# EPICS substitutions: wtrvac/Db/vac.substitutions
file "TP_AI.template" { pattern
{P,  		    SIG,	OFFS, TYP,    PREC,   EGU,   LOPR,  HOPR, H,	MAXVAL, PB_ADDR}
{CstatH-Vac:TP001,   MotV,	248,  BYTE,   0,      "V",   0,	100,	100,	100,	5}
{CstatH-Vac:TP001,   BearingT,	249,  BYTE,   0,      "°C",  0,	100,	100,	100,	5}
{CstatH-Vac:TP001,   PSupplyT,	250,  BYTE,   0,      "°C",  0,	100,	100,	100,	5}
{CstatH-Vac:TP001,   CPU_T,	251,  BYTE,   0,      "°C",  0,	100,	100,	100,	5}
{CstatH-Vac:TP001,   MotI,	256,  UINT16, 3,      "A",   0,	10,	10000,	10,	5}
{CstatH-Vac:TP001,   MotP,	258,  UINT16, 0,      "W",   0,	200,	200,	200,	5}
{CstatH-Vac:TP001,   MotPLimit,	260,  UINT16, 0,      "W",   0,	200,	200,	200,	5}
{CstatH-Vac:TP001,   Freq,	262,  UINT16, 0,      "Hz",  0,	1500,	1500,	1500,	5}
{CstatH-Vac:TP001,   FreqSP,	264,  UINT16, 0,      "Hz",  0,	1500,	1500,	1500,	5}
{CstatH-Vac:TP001,   NoOfStarts,266,  UINT16, 0,      "",    0,	65535,	65535,	65535,	5}
{CstatH-Vac:TP001,   LastOnTime,268,  UINT16, 0,      "min.",0,	65535,	65535,	65535,	5}
{CstatH-Vac:TP001,   OpTime,	270,  UINT16, 0,      "h",   0,	65535,	65535,	65535,	5}
}

file "TP_TD20.template" { pattern
{P,  			OFFS,	PB_ADDR}
{CstatH-Vac:TP002,   	278,  	6}
{CstatV-Vac:TP050,   	742,  	8}
{CstatV-Vac:TP060,   	906,  	9}
}

file "CtrlBitwRdBack.template" { pattern

{P,                   SIG,	S_OFFS, S_BIT, S_ZNAM, S_ONAM, C_OFFS, C_BIT, C_ZNAM,   C_ONAM,	INIT_EVNT}
{CstatH-Vac:TP002,    Remote,	276,	 7     Local,  Remote, 46,	  2,	 Local, Remote,	7}
{CstatV-Vac:TP050,    Remote,	740,	 7     Local,  Remote, 144,	  2,	 Local, Remote,	7}
{CstatV-Vac:TP060,    Remote,	904,	 7     Local,  Remote, 194,	  2,	 Local, Remote,	7}
#{CstatH-Vac:TP002,    On,	276,	 2     OFF,    ON,     47,	  0,	 Stop,  Start,	7}
}

file "ArcDet.template" { pattern
{SYS,	SUBS,	DEV,	  SIG,	    OFFS,	BIT,	ZNAM,	ONAM, DESC}
{HPRF,	Distr,	ArcDet01, cmdReset, 98,	0,	Idle,	Reset,	 "Reset Command"}
{HPRF,	Distr,	ArcDet01, cmdTest,  98,	1,	Idle,	Test, 	 "Test Command"}
{HPRF,	Distr,	ArcDet02, cmdReset, 98,	2,	Idle,	Reset,	 "Reset Command"}
{HPRF,	Distr,	ArcDet02, cmdTest,  98,	3,	Idle,	Test, 	 "Test Command"}
{HPRF,	Distr,	ArcDet03, cmdReset, 98,	4,	Idle,	Reset,	 "Reset Command"}
{HPRF,	Distr,	ArcDet03, cmdTest,  98,	5,	Idle,	Test, 	 "Test Command"}
{HPRF,	Distr,	ArcDet04, cmdReset, 98,	6,	Idle,	Reset,	 "Reset Command"}
{HPRF,	Distr,	ArcDet04, cmdTest,  98,	7,	Idle,	Test, 	 "Test Command"}
{HPRF,	Distr,	ArcDet05, cmdReset, 99,	0,	Idle,	Reset,	 "Reset Command"}
{HPRF,	Distr,	ArcDet05, cmdTest,  99,	1,	Idle,	Test, 	 "Test Command"}
{HPRF,	Distr,	ArcDet06, cmdReset, 99,	2,	Idle,	Reset,	 "Reset Command"}
{HPRF,	Distr,	ArcDet06, cmdTest,  99,	3,	Idle,	Test, 	 "Test Command"}
{HPRF,	Distr,	ArcDet07, cmdReset, 99,	4,	Idle,	Reset,	 "Reset Command"}
{HPRF,	Distr,	ArcDet07, cmdTest,  99,	5,	Idle,	Test, 	 "Test Command"}
}

file "Interlock.template" { pattern
{SYS,	SUBS,	DEV,	       OFFS1,	OFFS2, B0,	B1,	B2,	B3,	B4,	B5,	B6,	B7, INIT_EVNT}
{LLRF,	Cntrl,	SlowIntlk,     440, 	102, "FREIA bunker door closed", "FREIA bunker cleared", "PwrCoupler Wtr Cooling", "", "Mobile LLRF", "CM Cryogenics", "Software Interlock","Test", 7}
{HPRF,	SSA_A,	ExtIntlkHNOSS, 444, 	104, "RFSwitchBoard1 Path", "FREIA bunker cleared", "Wtr Flow Guard3", "Wtr Flow Guard4", "RFSwitchBoard2 Sw2", "RFSwitchBoard3 Sw1", "Watchdog-1","Test", 7}
{HPRF,	SSA_A,	ExtIntlkTest,  448, 	106, "RFSwitchBoard1 Sw9", "RFSwitchBoard1 Sw13", "Wtr Flow Guard3", "Wtr Flow Guard4", "RFSwitchBoard2 Sw1", "", "Watchdog-1","Test", 7}
{HPRF,	SSA_A,	ExtIntlkLoad2, 452, 	108, "RFSwitchBoard1 Sw9", "RFSwitchBoard1 Sw15", "Wtr Flow Guard5", "", "", "", "Watchdog-1","Test", 7}
{HPRF,	SSA_A,	ExtIntlkCM,    456, 	110, "RFSwitchBoard1 Path", "FREIA bunker cleared", "Wtr Flow Guard1", "Wtr Flow Guard2", "", "", "Watchdog-1","Test", 7}
{HPRF,	DBE,	ExtIntlkHNOSS, 460, 	112, "RFSwitchBoard1 Path", "RFSwitchBoard1 Sw14", "Wtr Flow Guard3", "Wtr Flow Guard4", "RFSwitchBoard2 Sw2", "RFSwitchBoard3 Sw1", "Watchdog-1","Test", 7}
{HPRF,	DBE,	ExtIntlkTest,  464, 	114, "RFSwitchBoard1 Sw12", "RFSwitchBoard1 Sw14", "Wtr Flow Guard3", "Wtr Flow Guard4", "RFSwitchBoard2 Sw1", "", "Watchdog-1","Test", 7}
{HPRF,	DBE,	ExtIntlkLoad2, 468, 	116, "RFSwitchBoard1 Sw12", "RFSwitchBoard1 Sw16", "Wtr Flow Guard5", "", "", "", "Watchdog-1","Test", 7}
{HPRF,	DBE,	ExtIntlkCM,    472, 	118, "RFSwitchBoard1 Path", "FREIA bunker cleared", "Wtr Flow Guard1", "Wtr Flow Guard2", "", "", "Watchdog-1","Test", 7}
{HPRF,	PwrCpl,	WtrCIntlk,     476, 	120, "TT01", "TT02", "TT03", "TT04", "Wtr Flow Guard7", "Wtr Flow Guard8", "FT03","FT04", 7}
{LLRF,	Mobile,	Intlk,         480, 	122, "FREIA bunker door closed", "FREIA bunker cleared", "", "", "", "", "","", 7}
{HPRF,	SSA_B,	ExtIntlkHNOSS, 484, 	124, "RFSwitchBoard1 Path", "FREIA bunker cleared", "Wtr Flow Guard3", "Wtr Flow Guard4", "RFSwitchBoard2 Sw2", "RFSwitchBoard3 Sw1", "Watchdog-1","Test", 7}
{HPRF,	SSA_B,	ExtIntlkTest,  488, 	126, "RFSwitchBoard1 Path", "", "Wtr Flow Guard3", "Wtr Flow Guard4", "RFSwitchBoard2 Sw1", "", "Watchdog-1","Test", 7}
{HPRF,	SSA_B,	ExtIntlkLoad2, 492, 	128, "RFSwitchBoard1 Path", "", "Wtr Flow Guard5", "", "", "", "Watchdog-1","Test", 7}
{HPRF,	SSA_B,	ExtIntlkCM,    496, 	130, "RFSwitchBoard1 Path", "FREIA bunker cleared", "Wtr Flow Guard1", "Wtr Flow Guard2", "", "", "Watchdog-1","Test", 7}
{HPRF,	SSA_A,	ExtIntlkCM2,  1070, 	244, "RFSwitchBoard1 Path", "FREIA bunker cleared", "Wtr Flow Guard3", "Wtr Flow Guard4", "RFSwitchBoard2 Sw2", "RFSwitchBoard3 Sw2", "Watchdog-1","Test", 7}
{HPRF,	DBE,	ExtIntlkCM2,  1074, 	246, "RFSwitchBoard1 Path", "FREIA bunker cleared", "Wtr Flow Guard3", "Wtr Flow Guard4", "RFSwitchBoard2 Sw2", "RFSwitchBoard3 Sw1", "Watchdog-1","Test", 7}
{HPRF,	SSA_B,	ExtIntlkCM2,  1078, 	248, "RFSwitchBoard1 Path", "FREIA bunker cleared", "Wtr Flow Guard3", "Wtr Flow Guard4", "RFSwitchBoard2 Sw2", "RFSwitchBoard3 Sw1", "Watchdog-1","Test", 7}
}

file "Dwtr_WFG.template" { pattern
{P,  		NR,	 OFFS,	B}
{WtrC-Dwtr,	01	 506	0}
{WtrC-Dwtr,	02	 506	1}
{WtrC-Dwtr,	03	 506	2}
{WtrC-Dwtr,	04	 506	3}
{WtrC-Dwtr,	05	 506	4}
{WtrC-Dwtr,	06	 506	5}
{WtrC-Dwtr,	07	 506	6}
{WtrC-Dwtr,	08	 506	7}
}

# ADC inputs

file "Dwtr_AIx4.template" { pattern
{P,  	 	    SIG,	OFFS,  STAT_OFFS, SHFT, LOPR,  HOPR EGU,  PREC}
{"Env-Bunker1:QT001", RdV,	514,   508        4,     0	25,   "%",2}
{"Env-CmpRoom:QT002", RdV,	518,   509        0,     0	25,   "%",2}
{"WtrC-Dwtr:PwrCpl-FT01", RdV,	528,   526        0,     0	50,   "l/h",2}
{"WtrC-Dwtr:PwrCpl-FT02", RdV,	532,   526        4,     0	50,   "l/h",2}
{"WtrC-Dwtr:PwrCpl-FT03", RdV,	536,   527        0,     0	50,   "l/h",2}
{"WtrC-Dwtr:PwrCpl-FT04", RdV,	540,   527        4,     0	50,   "l/h",2}
{"WtrC-Dwtr:PwrCpl-TT01", RdV,	546,   544        0,     0	50,   "ᵒC",1}
{"WtrC-Dwtr:PwrCpl-TT02", RdV,	550,   544        4,     0	50,   "ᵒC",1}
{"WtrC-Dwtr:PwrCpl-TT03", RdV,	554,   545        0,     0	50,   "ᵒC",1}
{"WtrC-Dwtr:PwrCpl-TT04", RdV,	558,   545        4,     0	50,   "ᵒC",1}
{"WtrC-Dwtr:Kly-FT01", 	  RdV,	564,   562        0,     0	500,  "l/h",2}
{"WtrC-Dwtr:Kly-FT02", 	  RdV,	568,   562        4,     0	10,   "l/h",2}
{"WtrC-Dwtr:Kly-FT03",	  RdV,	572,   563        0,     0	50,   "l/h",2}
{"WtrC-Dwtr:Kly-FT04", 	  RdV,	576,   563        4,     0	50,   "l/h",2}
}
